% RSLogix 500 project HEATER ANALOG CONTROL WITH PID.RSS, saved by version 8.30.00.16 %
PROJECT "UNTITLED"    % processor: Bul.1763 MicroLogix 1100 Series B %

PROGRAM FILES
  LAD 2 "MAIN"  4 rungs
  LAD 3 "IO"  4 rungs  % IO %
  LAD 4 "CONTROL"  1 rungs
  LAD 5 "ALARM"  4 rungs

DATA FILES
  O0 OUTPUT  9 elements
  I1 INPUT  16 elements
  S2 STATUS  66 elements
  B3 BINARY  1 elements
  T4 TIMER  1 elements
  C5 COUNTER  1 elements
  R6 CONTROL  1 elements
  N7 INTEGER  2 elements
  F8 FLOAT  1 elements
  PD9 TEMP  1 elements

LADDER 2 "MAIN"
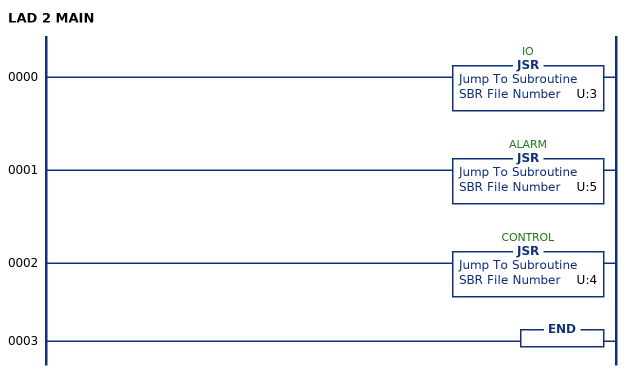
% Rung: 0 %  % edit flag set %
SOR JSR U:3 EOR
%   U:3  "IO" %
% Rung: 1 %  % edit flag set %
SOR JSR U:5 EOR
%   U:5  "ALARM" %
% Rung: 2 %  % edit flag set %
SOR JSR U:4 EOR
%   U:4  "CONTROL" %
% Rung: 3 %
SOR END EOR

LADDER 3 "IO"    % IO %
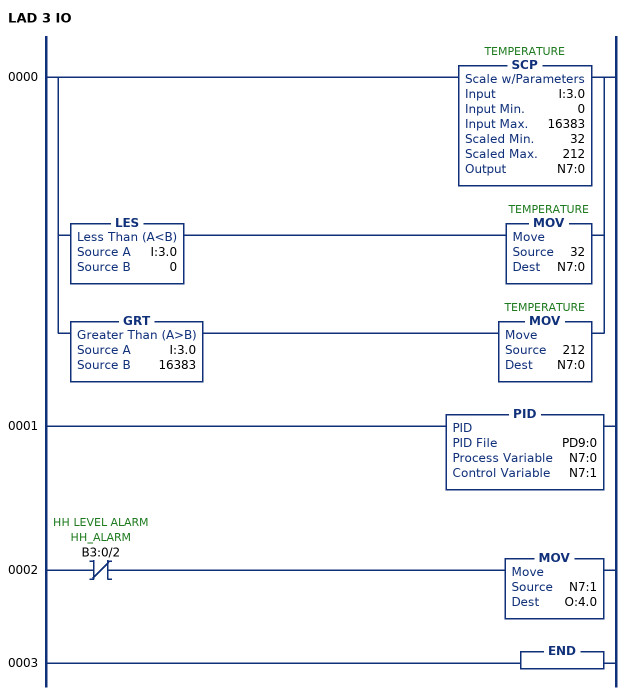
% Rung: 0 %
SOR BST SCP I:3.0 0 16383 32 212 N7:0 NXB LES I:3.0 0 MOV 32 N7:0 NXB GRT I:3.0 16383 MOV 212 N7:0 BND EOR
%   N7:0  "TEMPERATURE" %
% Rung: 1 %
SOR PID PD9:0 N7:0 N7:1 EOR
%   N7:0  "TEMPERATURE" %
%   N7:1  "PID OTPUT" %
% Rung: 2 %
SOR XIO B3:0/2 MOV N7:1 O:4.0 EOR
%   B3:0/2  HH_ALARM  "HH LEVEL ALARM" %
%   N7:1  "PID OTPUT" %
% Rung: 3 %
SOR END EOR

LADDER 5 "ALARM"
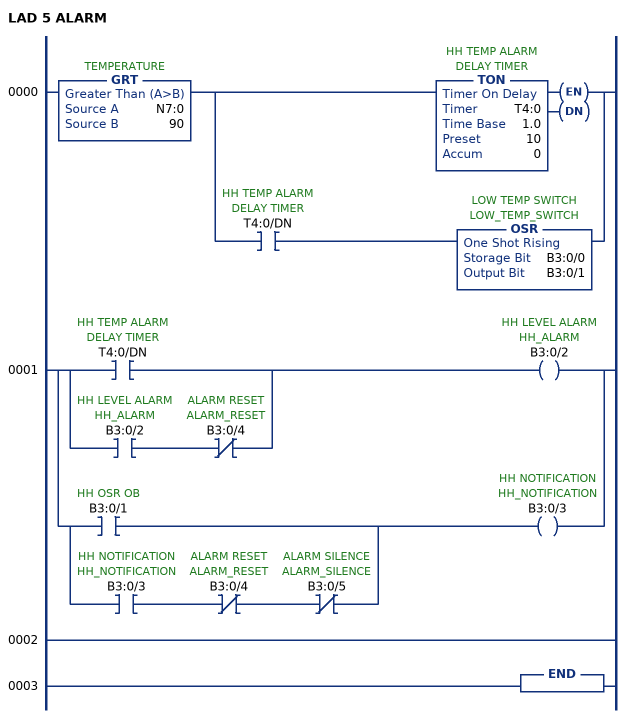
% Rung: 0 %  % edit flag set %
SOR GRT N7:0 90 BST TON T4:0 1.0 10 0 NXB XIC T4:0/DN OSR B3:0/0 B3:0/1 BND EOR
%   N7:0  "TEMPERATURE" %
%   T4:0  "HH TEMP ALARM DELAY TIMER" %
%   B3:0/0  LOW_TEMP_SWITCH  "LOW TEMP SWITCH" %
%   B3:0/1  "HH OSR OB" %
% Rung: 1 %  % edit flag set %
SOR BST BST XIC T4:0/DN NXB XIC B3:0/2 XIO B3:0/4 BND OTE B3:0/2 NXB BST XIC B3:0/1 NXB XIC B3:0/3 XIO B3:0/4 XIO B3:0/5 BND OTE B3:0/3 BND EOR
%   T4:0  "HH TEMP ALARM DELAY TIMER" %
%   B3:0/2  HH_ALARM  "HH LEVEL ALARM" %
%   B3:0/4  ALARM_RESET  "ALARM RESET" %
%   B3:0/1  "HH OSR OB" %
%   B3:0/3  HH_NOTIFICATION  "HH NOTIFICATION" %
%   B3:0/5  ALARM_SILENCE  "ALARM SILENCE" %
% Rung: 2 %  % edit flag set %
SOR EOR
% Rung: 3 %
SOR END EOR

OTHER DOCUMENTED ADDRESSES
  I:0.0/0  "LOW TEMP SWITCH INPUT"
  I:0.0/1  "HIGH TEM SWITCH INPUT"
  I:1.0/0  "LOW TEMP SWITCH INPUT"
  I:1.0/1  "HIGH TEMP SWITCH INPUT"
  I:3.0/0  "TEMP SENSOR INPUT"
  O:2.0/0  "HEATER OUTPUT"
  O:4.0/0  "TEMP CONTROLLER"
